// TIA Portal V17 export
// export: Created 2023-12-22T15:03:17.9510383Z, ExportSetting WithDefaults, DisplayName Totally Integrated Automation Portal, DisplayVersion V17, DisplayName TIA Portal Openness, DisplayVersion V17, DisplayName TIA Portal Version Control Interface, DisplayVersion V17, DisplayName STEP 7 Professional, DisplayVersion V17, DisplayName STEP 7 Safety, DisplayVersion V17, DisplayName WinCC Advanced, DisplayVersion V17
DATA_BLOCK "Route_Check_DB"   // DB8
VERSION : 0.1
// stored: AutoNumber true, DBAccessibleFromOPCUA true, DBAccessibleFromWebserver true, InstanceOfName Route_Check, InstanceOfType FB
"Route_Check"
   // VAR
   //    ready_2_7_from_2_9 : Bool;
   //    ready_2_7_from_SKV13 : Bool;
   //    ready_2_7_from_2_6_1 : Bool;
   //    ready_2_7_from_2_6_2 : Bool;
   //    ready_2_7_q_1 : Bool;
   //    ready_2_7_q_2 : Bool;
   //    ready_2_6_from_SKV14 : Bool;
   //    ready_2_6_from_2_5_1 : Bool;
   //    ready_2_6_from_2_5_2 : Bool;
   //    ready_2_6_q_1 : Bool;
   //    ready_2_6_q_2 : Bool;
   // END_VAR
BEGIN
END_DATA_BLOCK
